// TIA Portal V17 export
// export: Created 2023-02-13T11:16:45.7840585Z, ExportSetting WithDefaults, DisplayName Totally Integrated Automation Portal, DisplayVersion V17, DisplayName TIA Portal Openness, DisplayVersion V17, DisplayName TIA Portal Teamcenter Gateway, DisplayVersion V17, DisplayName TIA Portal Version Control Interface, DisplayVersion V17, DisplayName SINAMICS Startdrive Advanced, DisplayVersion V17, DisplayName SINAMICS Startdrive G130, G150, S120, S150, SINAMICS MV, S210, DisplayVersion V17, DisplayName SINAMICS Startdrive G110M, G120, G120C, G120D, G120P, G115D, DisplayVersion V17, DisplayName STEP 7 Professional, DisplayVersion V17, DisplayName STEP 7 Safety, DisplayVersion V17, DisplayName WinCC Professional, DisplayVersion V17
ORGANIZATION_BLOCK "Totalizer_OB"   // OB31, LAD, CyclicInterrupt
{ S7_Optimized_Access := 'TRUE' }
VERSION : 0.1
// stored: AutoNumber false, IsIECCheckEnabled false, SetENOAutomatically false
   VAR_INPUT
      Initial_Call : Bool;   // Initial call of this OB
      Event_Count : Int;   // Events discarded
   END_VAR
   VAR_TEMP   // added for the SCL form of the ladder/FBD networks
      _w1 : Bool;
   END_VAR
BEGIN

REGION Network 1: Totalizer FT-00.01 Process Water Control
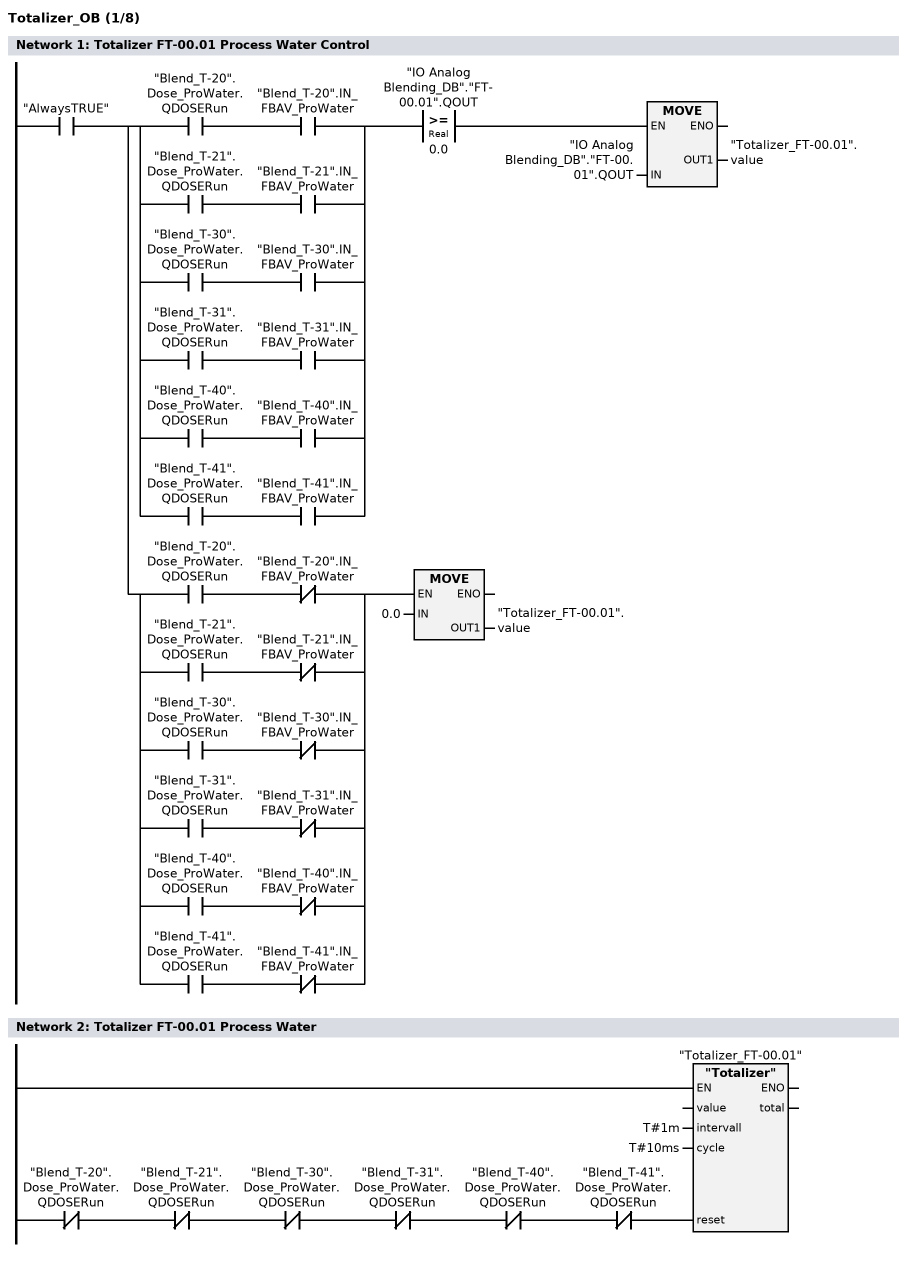
   RUNG wire#powerrail
      Contact( "AlwaysTRUE" )
      wire#w1
      Contact( "Blend_T-20".Dose_ProWater.QDOSERun )
      Contact( "Blend_T-20".IN_FBAV_ProWater )
      wire#w2
      { S7_Templates := "SrcType := Real" } GE_Contact(in1 := "IO Analog Blending_DB"."FT-00.01".QOUT, in2 := 0.0)
      Move(in := "IO Analog Blending_DB"."FT-00.01".QOUT, out1 => "Totalizer_FT-00.01".value)
   END_RUNG
   RUNG wire#w1
      Contact( "Blend_T-21".Dose_ProWater.QDOSERun )
      Contact( "Blend_T-21".IN_FBAV_ProWater )
   END_RUNG wire#w2
   RUNG wire#w1
      Contact( "Blend_T-30".Dose_ProWater.QDOSERun )
      Contact( "Blend_T-30".IN_FBAV_ProWater )
   END_RUNG wire#w2
   RUNG wire#w1
      Contact( "Blend_T-31".Dose_ProWater.QDOSERun )
      Contact( "Blend_T-31".IN_FBAV_ProWater )
   END_RUNG wire#w2
   RUNG wire#w1
      Contact( "Blend_T-40".Dose_ProWater.QDOSERun )
      Contact( "Blend_T-40".IN_FBAV_ProWater )
   END_RUNG wire#w2
   RUNG wire#w1
      Contact( "Blend_T-41".Dose_ProWater.QDOSERun )
      Contact( "Blend_T-41".IN_FBAV_ProWater )
   END_RUNG wire#w2
   RUNG wire#w1
      Contact( "Blend_T-20".Dose_ProWater.QDOSERun )
      I_Contact( "Blend_T-20".IN_FBAV_ProWater )
      wire#w3
      Move(in := 0.0, out1 => "Totalizer_FT-00.01".value)
   END_RUNG
   RUNG wire#w1
      Contact( "Blend_T-21".Dose_ProWater.QDOSERun )
      I_Contact( "Blend_T-21".IN_FBAV_ProWater )
   END_RUNG wire#w3
   RUNG wire#w1
      Contact( "Blend_T-30".Dose_ProWater.QDOSERun )
      I_Contact( "Blend_T-30".IN_FBAV_ProWater )
   END_RUNG wire#w3
   RUNG wire#w1
      Contact( "Blend_T-31".Dose_ProWater.QDOSERun )
      I_Contact( "Blend_T-31".IN_FBAV_ProWater )
   END_RUNG wire#w3
   RUNG wire#w1
      Contact( "Blend_T-40".Dose_ProWater.QDOSERun )
      I_Contact( "Blend_T-40".IN_FBAV_ProWater )
   END_RUNG wire#w3
   RUNG wire#w1
      Contact( "Blend_T-41".Dose_ProWater.QDOSERun )
      I_Contact( "Blend_T-41".IN_FBAV_ProWater )
   END_RUNG wire#w3
   // the same network as SCL:
   IF "AlwaysTRUE" AND (("Blend_T-20".Dose_ProWater.QDOSERun AND "Blend_T-20".IN_FBAV_ProWater) OR ("Blend_T-21".Dose_ProWater.QDOSERun AND "Blend_T-21".IN_FBAV_ProWater) OR ("Blend_T-30".Dose_ProWater.QDOSERun AND "Blend_T-30".IN_FBAV_ProWater) OR ("Blend_T-31".Dose_ProWater.QDOSERun AND "Blend_T-31".IN_FBAV_ProWater) OR ("Blend_T-40".Dose_ProWater.QDOSERun AND "Blend_T-40".IN_FBAV_ProWater) OR ("Blend_T-41".Dose_ProWater.QDOSERun AND "Blend_T-41".IN_FBAV_ProWater)) AND ("IO Analog Blending_DB"."FT-00.01".QOUT >= 0.0) THEN
       "Totalizer_FT-00.01".value := "IO Analog Blending_DB"."FT-00.01".QOUT;
   END_IF;
   IF "AlwaysTRUE" AND (("Blend_T-20".Dose_ProWater.QDOSERun AND NOT "Blend_T-20".IN_FBAV_ProWater) OR ("Blend_T-21".Dose_ProWater.QDOSERun AND NOT "Blend_T-21".IN_FBAV_ProWater) OR ("Blend_T-30".Dose_ProWater.QDOSERun AND NOT "Blend_T-30".IN_FBAV_ProWater) OR ("Blend_T-31".Dose_ProWater.QDOSERun AND NOT "Blend_T-31".IN_FBAV_ProWater) OR ("Blend_T-40".Dose_ProWater.QDOSERun AND NOT "Blend_T-40".IN_FBAV_ProWater) OR ("Blend_T-41".Dose_ProWater.QDOSERun AND NOT "Blend_T-41".IN_FBAV_ProWater)) THEN
       "Totalizer_FT-00.01".value := 0.0;
   END_IF;
END_REGION

REGION Network 2: Totalizer FT-00.01 Process Water
   RUNG wire#powerrail
      "Totalizer_FT-00.01"(reset := wire#w1, value :=, intervall := T#1m, cycle := T#10ms, total =>)
   END_RUNG
   RUNG wire#powerrail
      I_Contact( "Blend_T-20".Dose_ProWater.QDOSERun )
      I_Contact( "Blend_T-21".Dose_ProWater.QDOSERun )
      I_Contact( "Blend_T-30".Dose_ProWater.QDOSERun )
      I_Contact( "Blend_T-31".Dose_ProWater.QDOSERun )
      I_Contact( "Blend_T-40".Dose_ProWater.QDOSERun )
      I_Contact( "Blend_T-41".Dose_ProWater.QDOSERun )
   END_RUNG wire#w1
   // the same network as SCL:
   "Totalizer_FT-00.01"(intervall := T#1m,   // "Totalizer"
                        cycle := T#10ms,
                        reset := NOT "Blend_T-20".Dose_ProWater.QDOSERun AND NOT "Blend_T-21".Dose_ProWater.QDOSERun AND NOT "Blend_T-30".Dose_ProWater.QDOSERun AND NOT "Blend_T-31".Dose_ProWater.QDOSERun AND NOT "Blend_T-40".Dose_ProWater.QDOSERun AND NOT "Blend_T-41".Dose_ProWater.QDOSERun);
END_REGION

REGION Network 4: Totalizer FT.02.01 Chili Awetan 1 Control
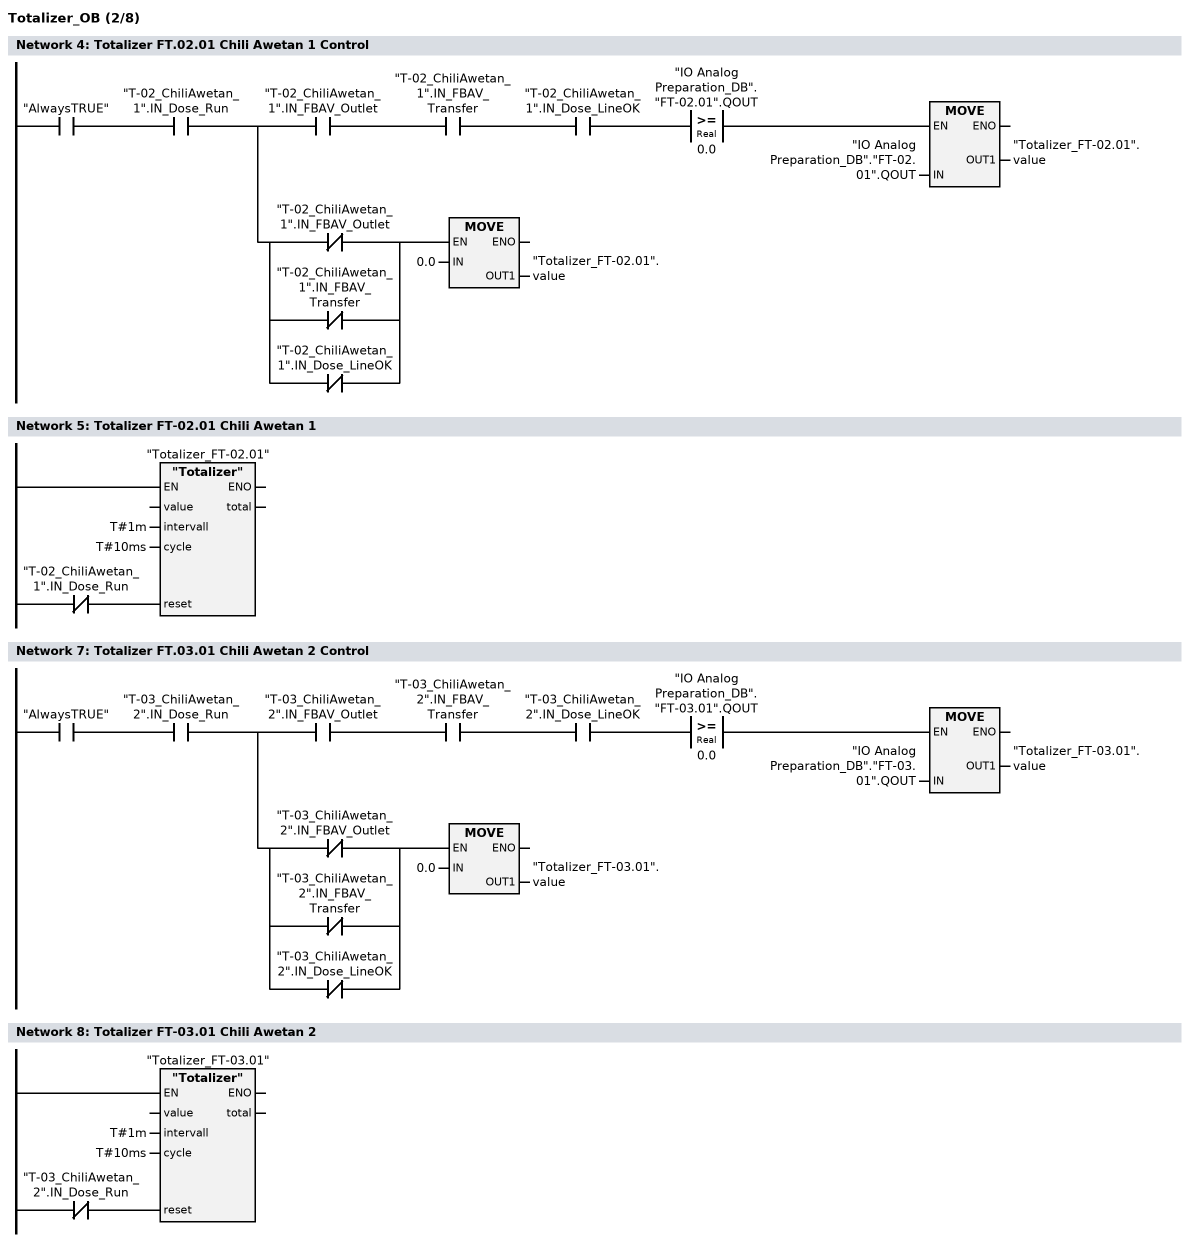
   RUNG wire#powerrail
      Contact( "AlwaysTRUE" )
      Contact( "T-02_ChiliAwetan_1".IN_Dose_Run )
      wire#w1
      Contact( "T-02_ChiliAwetan_1".IN_FBAV_Outlet )
      Contact( "T-02_ChiliAwetan_1".IN_FBAV_Transfer )
      Contact( "T-02_ChiliAwetan_1".IN_Dose_LineOK )
      { S7_Templates := "SrcType := Real" } GE_Contact(in1 := "IO Analog Preparation_DB"."FT-02.01".QOUT, in2 := 0.0)
      Move(in := "IO Analog Preparation_DB"."FT-02.01".QOUT, out1 => "Totalizer_FT-02.01".value)
   END_RUNG
   RUNG wire#w1
      I_Contact( "T-02_ChiliAwetan_1".IN_FBAV_Outlet )
      wire#w2
      Move(in := 0.0, out1 => "Totalizer_FT-02.01".value)
   END_RUNG
   RUNG wire#w1
      I_Contact( "T-02_ChiliAwetan_1".IN_FBAV_Transfer )
   END_RUNG wire#w2
   RUNG wire#w1
      I_Contact( "T-02_ChiliAwetan_1".IN_Dose_LineOK )
   END_RUNG wire#w2
   // the same network as SCL:
   #_w1 := "AlwaysTRUE" AND "T-02_ChiliAwetan_1".IN_Dose_Run;
   IF #_w1 AND "T-02_ChiliAwetan_1".IN_FBAV_Outlet AND "T-02_ChiliAwetan_1".IN_FBAV_Transfer AND "T-02_ChiliAwetan_1".IN_Dose_LineOK AND ("IO Analog Preparation_DB"."FT-02.01".QOUT >= 0.0) THEN
       "Totalizer_FT-02.01".value := "IO Analog Preparation_DB"."FT-02.01".QOUT;
   END_IF;
   IF #_w1 AND (NOT "T-02_ChiliAwetan_1".IN_FBAV_Outlet OR NOT "T-02_ChiliAwetan_1".IN_FBAV_Transfer OR NOT "T-02_ChiliAwetan_1".IN_Dose_LineOK) THEN
       "Totalizer_FT-02.01".value := 0.0;
   END_IF;
END_REGION

REGION Network 5: Totalizer FT-02.01 Chili Awetan 1
   RUNG wire#powerrail
      "Totalizer_FT-02.01"(reset := wire#w1, value :=, intervall := T#1m, cycle := T#10ms, total =>)
   END_RUNG
   RUNG wire#powerrail
      I_Contact( "T-02_ChiliAwetan_1".IN_Dose_Run )
   END_RUNG wire#w1
   // the same network as SCL:
   "Totalizer_FT-02.01"(intervall := T#1m, cycle := T#10ms, reset := NOT "T-02_ChiliAwetan_1".IN_Dose_Run);   // "Totalizer"
END_REGION

REGION Network 7: Totalizer FT.03.01 Chili Awetan 2 Control
   RUNG wire#powerrail
      Contact( "AlwaysTRUE" )
      Contact( "T-03_ChiliAwetan_2".IN_Dose_Run )
      wire#w1
      Contact( "T-03_ChiliAwetan_2".IN_FBAV_Outlet )
      Contact( "T-03_ChiliAwetan_2".IN_FBAV_Transfer )
      Contact( "T-03_ChiliAwetan_2".IN_Dose_LineOK )
      { S7_Templates := "SrcType := Real" } GE_Contact(in1 := "IO Analog Preparation_DB"."FT-03.01".QOUT, in2 := 0.0)
      Move(in := "IO Analog Preparation_DB"."FT-03.01".QOUT, out1 => "Totalizer_FT-03.01".value)
   END_RUNG
   RUNG wire#w1
      I_Contact( "T-03_ChiliAwetan_2".IN_FBAV_Outlet )
      wire#w2
      Move(in := 0.0, out1 => "Totalizer_FT-03.01".value)
   END_RUNG
   RUNG wire#w1
      I_Contact( "T-03_ChiliAwetan_2".IN_FBAV_Transfer )
   END_RUNG wire#w2
   RUNG wire#w1
      I_Contact( "T-03_ChiliAwetan_2".IN_Dose_LineOK )
   END_RUNG wire#w2
   // the same network as SCL:
   #_w1 := "AlwaysTRUE" AND "T-03_ChiliAwetan_2".IN_Dose_Run;
   IF #_w1 AND "T-03_ChiliAwetan_2".IN_FBAV_Outlet AND "T-03_ChiliAwetan_2".IN_FBAV_Transfer AND "T-03_ChiliAwetan_2".IN_Dose_LineOK AND ("IO Analog Preparation_DB"."FT-03.01".QOUT >= 0.0) THEN
       "Totalizer_FT-03.01".value := "IO Analog Preparation_DB"."FT-03.01".QOUT;
   END_IF;
   IF #_w1 AND (NOT "T-03_ChiliAwetan_2".IN_FBAV_Outlet OR NOT "T-03_ChiliAwetan_2".IN_FBAV_Transfer OR NOT "T-03_ChiliAwetan_2".IN_Dose_LineOK) THEN
       "Totalizer_FT-03.01".value := 0.0;
   END_IF;
END_REGION

REGION Network 8: Totalizer FT-03.01 Chili Awetan 2
   RUNG wire#powerrail
      "Totalizer_FT-03.01"(reset := wire#w1, value :=, intervall := T#1m, cycle := T#10ms, total =>)
   END_RUNG
   RUNG wire#powerrail
      I_Contact( "T-03_ChiliAwetan_2".IN_Dose_Run )
   END_RUNG wire#w1
   // the same network as SCL:
   "Totalizer_FT-03.01"(intervall := T#1m, cycle := T#10ms, reset := NOT "T-03_ChiliAwetan_2".IN_Dose_Run);   // "Totalizer"
END_REGION

REGION Network 10: Totalizer FT.04.01 Chili Awetan 3 Control
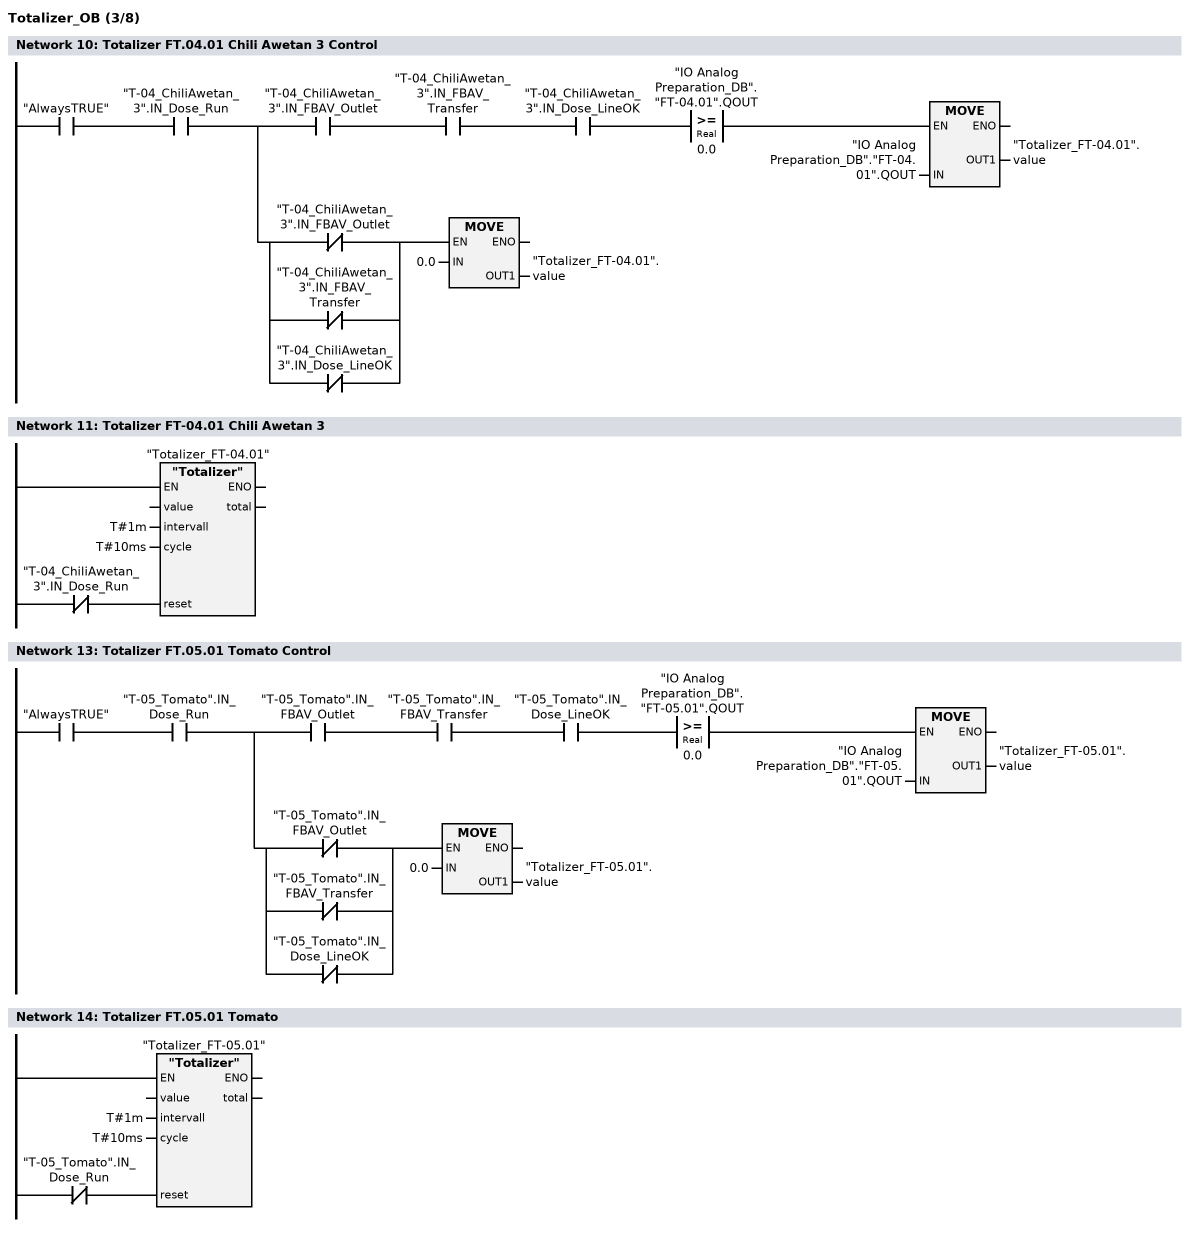
   RUNG wire#powerrail
      Contact( "AlwaysTRUE" )
      Contact( "T-04_ChiliAwetan_3".IN_Dose_Run )
      wire#w1
      Contact( "T-04_ChiliAwetan_3".IN_FBAV_Outlet )
      Contact( "T-04_ChiliAwetan_3".IN_FBAV_Transfer )
      Contact( "T-04_ChiliAwetan_3".IN_Dose_LineOK )
      { S7_Templates := "SrcType := Real" } GE_Contact(in1 := "IO Analog Preparation_DB"."FT-04.01".QOUT, in2 := 0.0)
      Move(in := "IO Analog Preparation_DB"."FT-04.01".QOUT, out1 => "Totalizer_FT-04.01".value)
   END_RUNG
   RUNG wire#w1
      I_Contact( "T-04_ChiliAwetan_3".IN_FBAV_Outlet )
      wire#w2
      Move(in := 0.0, out1 => "Totalizer_FT-04.01".value)
   END_RUNG
   RUNG wire#w1
      I_Contact( "T-04_ChiliAwetan_3".IN_FBAV_Transfer )
   END_RUNG wire#w2
   RUNG wire#w1
      I_Contact( "T-04_ChiliAwetan_3".IN_Dose_LineOK )
   END_RUNG wire#w2
   // the same network as SCL:
   #_w1 := "AlwaysTRUE" AND "T-04_ChiliAwetan_3".IN_Dose_Run;
   IF #_w1 AND "T-04_ChiliAwetan_3".IN_FBAV_Outlet AND "T-04_ChiliAwetan_3".IN_FBAV_Transfer AND "T-04_ChiliAwetan_3".IN_Dose_LineOK AND ("IO Analog Preparation_DB"."FT-04.01".QOUT >= 0.0) THEN
       "Totalizer_FT-04.01".value := "IO Analog Preparation_DB"."FT-04.01".QOUT;
   END_IF;
   IF #_w1 AND (NOT "T-04_ChiliAwetan_3".IN_FBAV_Outlet OR NOT "T-04_ChiliAwetan_3".IN_FBAV_Transfer OR NOT "T-04_ChiliAwetan_3".IN_Dose_LineOK) THEN
       "Totalizer_FT-04.01".value := 0.0;
   END_IF;
END_REGION

REGION Network 11: Totalizer FT-04.01 Chili Awetan 3
   RUNG wire#powerrail
      "Totalizer_FT-04.01"(reset := wire#w1, value :=, intervall := T#1m, cycle := T#10ms, total =>)
   END_RUNG
   RUNG wire#powerrail
      I_Contact( "T-04_ChiliAwetan_3".IN_Dose_Run )
   END_RUNG wire#w1
   // the same network as SCL:
   "Totalizer_FT-04.01"(intervall := T#1m, cycle := T#10ms, reset := NOT "T-04_ChiliAwetan_3".IN_Dose_Run);   // "Totalizer"
END_REGION

REGION Network 13: Totalizer FT.05.01 Tomato Control
   RUNG wire#powerrail
      Contact( "AlwaysTRUE" )
      Contact( "T-05_Tomato".IN_Dose_Run )
      wire#w1
      Contact( "T-05_Tomato".IN_FBAV_Outlet )
      Contact( "T-05_Tomato".IN_FBAV_Transfer )
      Contact( "T-05_Tomato".IN_Dose_LineOK )
      { S7_Templates := "SrcType := Real" } GE_Contact(in1 := "IO Analog Preparation_DB"."FT-05.01".QOUT, in2 := 0.0)
      Move(in := "IO Analog Preparation_DB"."FT-05.01".QOUT, out1 => "Totalizer_FT-05.01".value)
   END_RUNG
   RUNG wire#w1
      I_Contact( "T-05_Tomato".IN_FBAV_Outlet )
      wire#w2
      Move(in := 0.0, out1 => "Totalizer_FT-05.01".value)
   END_RUNG
   RUNG wire#w1
      I_Contact( "T-05_Tomato".IN_FBAV_Transfer )
   END_RUNG wire#w2
   RUNG wire#w1
      I_Contact( "T-05_Tomato".IN_Dose_LineOK )
   END_RUNG wire#w2
   // the same network as SCL:
   #_w1 := "AlwaysTRUE" AND "T-05_Tomato".IN_Dose_Run;
   IF #_w1 AND "T-05_Tomato".IN_FBAV_Outlet AND "T-05_Tomato".IN_FBAV_Transfer AND "T-05_Tomato".IN_Dose_LineOK AND ("IO Analog Preparation_DB"."FT-05.01".QOUT >= 0.0) THEN
       "Totalizer_FT-05.01".value := "IO Analog Preparation_DB"."FT-05.01".QOUT;
   END_IF;
   IF #_w1 AND (NOT "T-05_Tomato".IN_FBAV_Outlet OR NOT "T-05_Tomato".IN_FBAV_Transfer OR NOT "T-05_Tomato".IN_Dose_LineOK) THEN
       "Totalizer_FT-05.01".value := 0.0;
   END_IF;
END_REGION

REGION Network 14: Totalizer FT.05.01 Tomato
   RUNG wire#powerrail
      "Totalizer_FT-05.01"(reset := wire#w1, value :=, intervall := T#1m, cycle := T#10ms, total =>)
   END_RUNG
   RUNG wire#powerrail
      I_Contact( "T-05_Tomato".IN_Dose_Run )
   END_RUNG wire#w1
   // the same network as SCL:
   "Totalizer_FT-05.01"(intervall := T#1m, cycle := T#10ms, reset := NOT "T-05_Tomato".IN_Dose_Run);   // "Totalizer"
END_REGION

REGION Network 16: Totalizer FT.06.01 Chili Fresh 1 Control
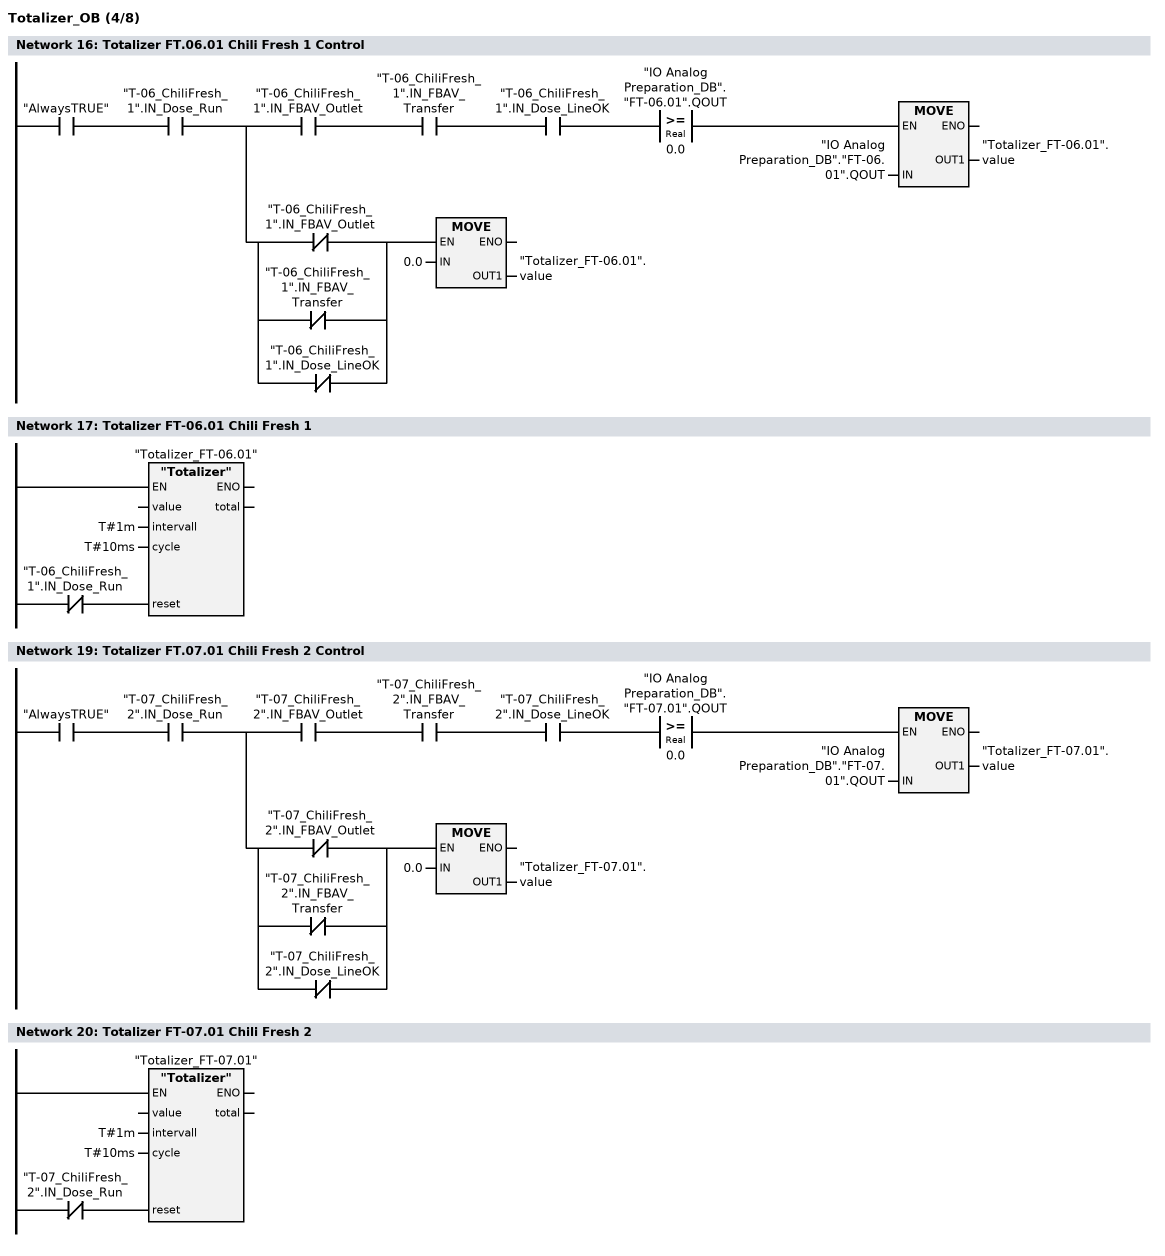
   RUNG wire#powerrail
      Contact( "AlwaysTRUE" )
      Contact( "T-06_ChiliFresh_1".IN_Dose_Run )
      wire#w1
      Contact( "T-06_ChiliFresh_1".IN_FBAV_Outlet )
      Contact( "T-06_ChiliFresh_1".IN_FBAV_Transfer )
      Contact( "T-06_ChiliFresh_1".IN_Dose_LineOK )
      { S7_Templates := "SrcType := Real" } GE_Contact(in1 := "IO Analog Preparation_DB"."FT-06.01".QOUT, in2 := 0.0)
      Move(in := "IO Analog Preparation_DB"."FT-06.01".QOUT, out1 => "Totalizer_FT-06.01".value)
   END_RUNG
   RUNG wire#w1
      I_Contact( "T-06_ChiliFresh_1".IN_FBAV_Outlet )
      wire#w2
      Move(in := 0.0, out1 => "Totalizer_FT-06.01".value)
   END_RUNG
   RUNG wire#w1
      I_Contact( "T-06_ChiliFresh_1".IN_FBAV_Transfer )
   END_RUNG wire#w2
   RUNG wire#w1
      I_Contact( "T-06_ChiliFresh_1".IN_Dose_LineOK )
   END_RUNG wire#w2
   // the same network as SCL:
   #_w1 := "AlwaysTRUE" AND "T-06_ChiliFresh_1".IN_Dose_Run;
   IF #_w1 AND "T-06_ChiliFresh_1".IN_FBAV_Outlet AND "T-06_ChiliFresh_1".IN_FBAV_Transfer AND "T-06_ChiliFresh_1".IN_Dose_LineOK AND ("IO Analog Preparation_DB"."FT-06.01".QOUT >= 0.0) THEN
       "Totalizer_FT-06.01".value := "IO Analog Preparation_DB"."FT-06.01".QOUT;
   END_IF;
   IF #_w1 AND (NOT "T-06_ChiliFresh_1".IN_FBAV_Outlet OR NOT "T-06_ChiliFresh_1".IN_FBAV_Transfer OR NOT "T-06_ChiliFresh_1".IN_Dose_LineOK) THEN
       "Totalizer_FT-06.01".value := 0.0;
   END_IF;
END_REGION

REGION Network 17: Totalizer FT-06.01 Chili Fresh 1
   RUNG wire#powerrail
      "Totalizer_FT-06.01"(reset := wire#w1, value :=, intervall := T#1m, cycle := T#10ms, total =>)
   END_RUNG
   RUNG wire#powerrail
      I_Contact( "T-06_ChiliFresh_1".IN_Dose_Run )
   END_RUNG wire#w1
   // the same network as SCL:
   "Totalizer_FT-06.01"(intervall := T#1m, cycle := T#10ms, reset := NOT "T-06_ChiliFresh_1".IN_Dose_Run);   // "Totalizer"
END_REGION

REGION Network 19: Totalizer FT.07.01 Chili Fresh 2 Control
   RUNG wire#powerrail
      Contact( "AlwaysTRUE" )
      Contact( "T-07_ChiliFresh_2".IN_Dose_Run )
      wire#w1
      Contact( "T-07_ChiliFresh_2".IN_FBAV_Outlet )
      Contact( "T-07_ChiliFresh_2".IN_FBAV_Transfer )
      Contact( "T-07_ChiliFresh_2".IN_Dose_LineOK )
      { S7_Templates := "SrcType := Real" } GE_Contact(in1 := "IO Analog Preparation_DB"."FT-07.01".QOUT, in2 := 0.0)
      Move(in := "IO Analog Preparation_DB"."FT-07.01".QOUT, out1 => "Totalizer_FT-07.01".value)
   END_RUNG
   RUNG wire#w1
      I_Contact( "T-07_ChiliFresh_2".IN_FBAV_Outlet )
      wire#w2
      Move(in := 0.0, out1 => "Totalizer_FT-07.01".value)
   END_RUNG
   RUNG wire#w1
      I_Contact( "T-07_ChiliFresh_2".IN_FBAV_Transfer )
   END_RUNG wire#w2
   RUNG wire#w1
      I_Contact( "T-07_ChiliFresh_2".IN_Dose_LineOK )
   END_RUNG wire#w2
   // the same network as SCL:
   #_w1 := "AlwaysTRUE" AND "T-07_ChiliFresh_2".IN_Dose_Run;
   IF #_w1 AND "T-07_ChiliFresh_2".IN_FBAV_Outlet AND "T-07_ChiliFresh_2".IN_FBAV_Transfer AND "T-07_ChiliFresh_2".IN_Dose_LineOK AND ("IO Analog Preparation_DB"."FT-07.01".QOUT >= 0.0) THEN
       "Totalizer_FT-07.01".value := "IO Analog Preparation_DB"."FT-07.01".QOUT;
   END_IF;
   IF #_w1 AND (NOT "T-07_ChiliFresh_2".IN_FBAV_Outlet OR NOT "T-07_ChiliFresh_2".IN_FBAV_Transfer OR NOT "T-07_ChiliFresh_2".IN_Dose_LineOK) THEN
       "Totalizer_FT-07.01".value := 0.0;
   END_IF;
END_REGION

REGION Network 20: Totalizer FT-07.01 Chili Fresh 2
   RUNG wire#powerrail
      "Totalizer_FT-07.01"(reset := wire#w1, value :=, intervall := T#1m, cycle := T#10ms, total =>)
   END_RUNG
   RUNG wire#powerrail
      I_Contact( "T-07_ChiliFresh_2".IN_Dose_Run )
   END_RUNG wire#w1
   // the same network as SCL:
   "Totalizer_FT-07.01"(intervall := T#1m, cycle := T#10ms, reset := NOT "T-07_ChiliFresh_2".IN_Dose_Run);   // "Totalizer"
END_REGION

REGION Network 22: Totalizer FT.08.01 Chili Fresh 3 Control
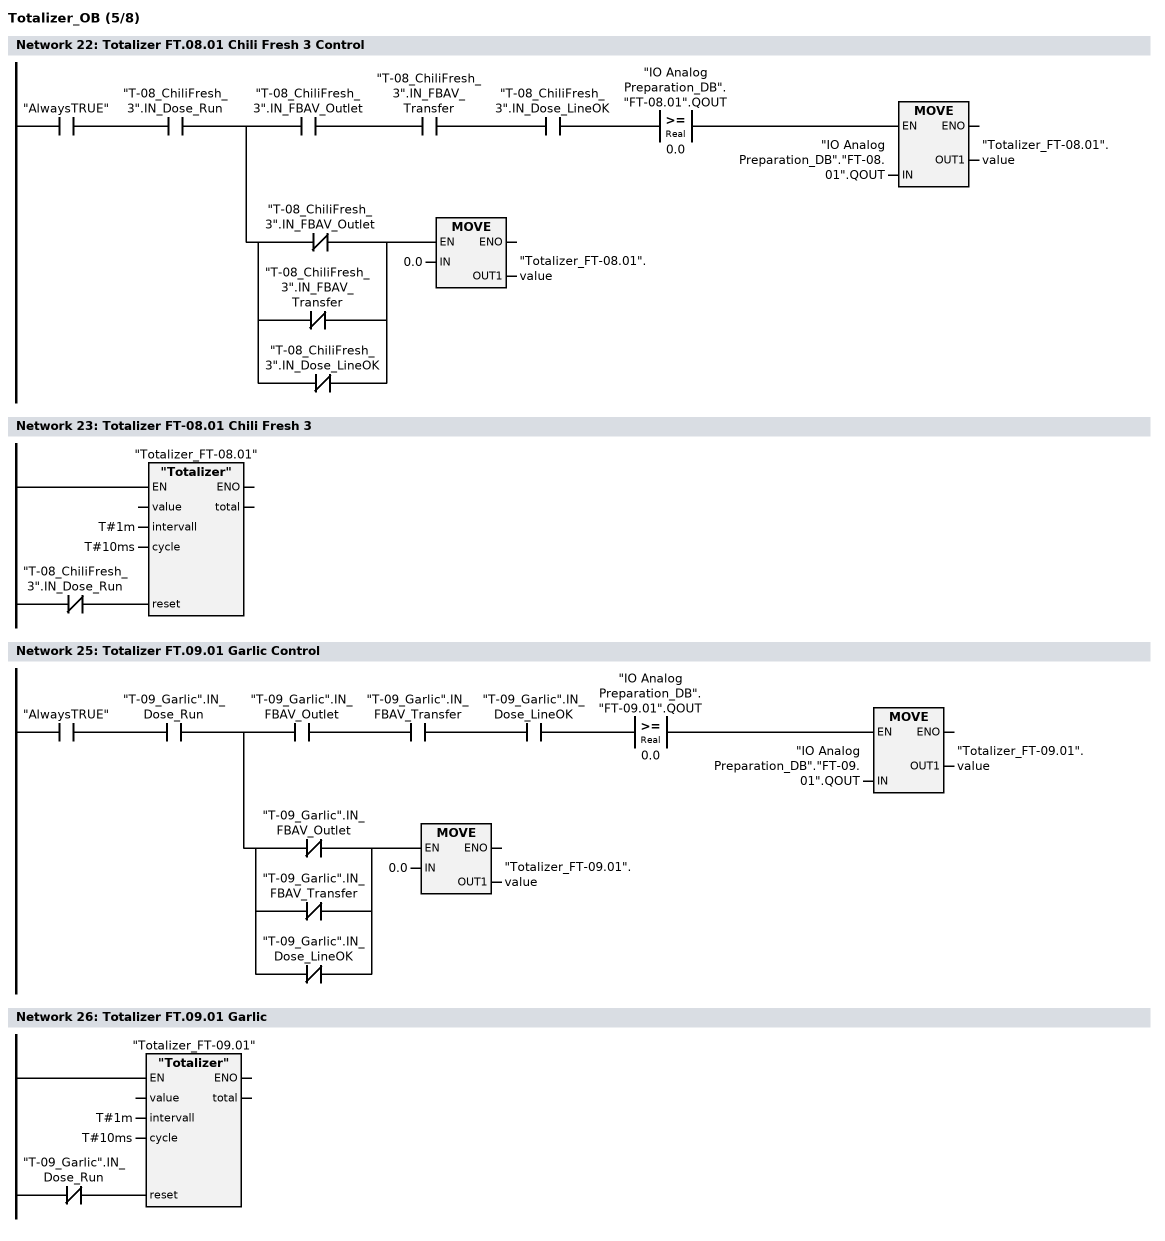
   RUNG wire#powerrail
      Contact( "AlwaysTRUE" )
      Contact( "T-08_ChiliFresh_3".IN_Dose_Run )
      wire#w1
      Contact( "T-08_ChiliFresh_3".IN_FBAV_Outlet )
      Contact( "T-08_ChiliFresh_3".IN_FBAV_Transfer )
      Contact( "T-08_ChiliFresh_3".IN_Dose_LineOK )
      { S7_Templates := "SrcType := Real" } GE_Contact(in1 := "IO Analog Preparation_DB"."FT-08.01".QOUT, in2 := 0.0)
      Move(in := "IO Analog Preparation_DB"."FT-08.01".QOUT, out1 => "Totalizer_FT-08.01".value)
   END_RUNG
   RUNG wire#w1
      I_Contact( "T-08_ChiliFresh_3".IN_FBAV_Outlet )
      wire#w2
      Move(in := 0.0, out1 => "Totalizer_FT-08.01".value)
   END_RUNG
   RUNG wire#w1
      I_Contact( "T-08_ChiliFresh_3".IN_FBAV_Transfer )
   END_RUNG wire#w2
   RUNG wire#w1
      I_Contact( "T-08_ChiliFresh_3".IN_Dose_LineOK )
   END_RUNG wire#w2
   // the same network as SCL:
   #_w1 := "AlwaysTRUE" AND "T-08_ChiliFresh_3".IN_Dose_Run;
   IF #_w1 AND "T-08_ChiliFresh_3".IN_FBAV_Outlet AND "T-08_ChiliFresh_3".IN_FBAV_Transfer AND "T-08_ChiliFresh_3".IN_Dose_LineOK AND ("IO Analog Preparation_DB"."FT-08.01".QOUT >= 0.0) THEN
       "Totalizer_FT-08.01".value := "IO Analog Preparation_DB"."FT-08.01".QOUT;
   END_IF;
   IF #_w1 AND (NOT "T-08_ChiliFresh_3".IN_FBAV_Outlet OR NOT "T-08_ChiliFresh_3".IN_FBAV_Transfer OR NOT "T-08_ChiliFresh_3".IN_Dose_LineOK) THEN
       "Totalizer_FT-08.01".value := 0.0;
   END_IF;
END_REGION

REGION Network 23: Totalizer FT-08.01 Chili Fresh 3
   RUNG wire#powerrail
      "Totalizer_FT-08.01"(reset := wire#w1, value :=, intervall := T#1m, cycle := T#10ms, total =>)
   END_RUNG
   RUNG wire#powerrail
      I_Contact( "T-08_ChiliFresh_3".IN_Dose_Run )
   END_RUNG wire#w1
   // the same network as SCL:
   "Totalizer_FT-08.01"(intervall := T#1m, cycle := T#10ms, reset := NOT "T-08_ChiliFresh_3".IN_Dose_Run);   // "Totalizer"
END_REGION

REGION Network 25: Totalizer FT.09.01 Garlic Control
   RUNG wire#powerrail
      Contact( "AlwaysTRUE" )
      Contact( "T-09_Garlic".IN_Dose_Run )
      wire#w1
      Contact( "T-09_Garlic".IN_FBAV_Outlet )
      Contact( "T-09_Garlic".IN_FBAV_Transfer )
      Contact( "T-09_Garlic".IN_Dose_LineOK )
      { S7_Templates := "SrcType := Real" } GE_Contact(in1 := "IO Analog Preparation_DB"."FT-09.01".QOUT, in2 := 0.0)
      Move(in := "IO Analog Preparation_DB"."FT-09.01".QOUT, out1 => "Totalizer_FT-09.01".value)
   END_RUNG
   RUNG wire#w1
      I_Contact( "T-09_Garlic".IN_FBAV_Outlet )
      wire#w2
      Move(in := 0.0, out1 => "Totalizer_FT-09.01".value)
   END_RUNG
   RUNG wire#w1
      I_Contact( "T-09_Garlic".IN_FBAV_Transfer )
   END_RUNG wire#w2
   RUNG wire#w1
      I_Contact( "T-09_Garlic".IN_Dose_LineOK )
   END_RUNG wire#w2
   // the same network as SCL:
   #_w1 := "AlwaysTRUE" AND "T-09_Garlic".IN_Dose_Run;
   IF #_w1 AND "T-09_Garlic".IN_FBAV_Outlet AND "T-09_Garlic".IN_FBAV_Transfer AND "T-09_Garlic".IN_Dose_LineOK AND ("IO Analog Preparation_DB"."FT-09.01".QOUT >= 0.0) THEN
       "Totalizer_FT-09.01".value := "IO Analog Preparation_DB"."FT-09.01".QOUT;
   END_IF;
   IF #_w1 AND (NOT "T-09_Garlic".IN_FBAV_Outlet OR NOT "T-09_Garlic".IN_FBAV_Transfer OR NOT "T-09_Garlic".IN_Dose_LineOK) THEN
       "Totalizer_FT-09.01".value := 0.0;
   END_IF;
END_REGION

REGION Network 26: Totalizer FT.09.01 Garlic
   RUNG wire#powerrail
      "Totalizer_FT-09.01"(reset := wire#w1, value :=, intervall := T#1m, cycle := T#10ms, total =>)
   END_RUNG
   RUNG wire#powerrail
      I_Contact( "T-09_Garlic".IN_Dose_Run )
   END_RUNG wire#w1
   // the same network as SCL:
   "Totalizer_FT-09.01"(intervall := T#1m, cycle := T#10ms, reset := NOT "T-09_Garlic".IN_Dose_Run);   // "Totalizer"
END_REGION

REGION Network 28: Totalizer FT.10.01 Vinegar Control
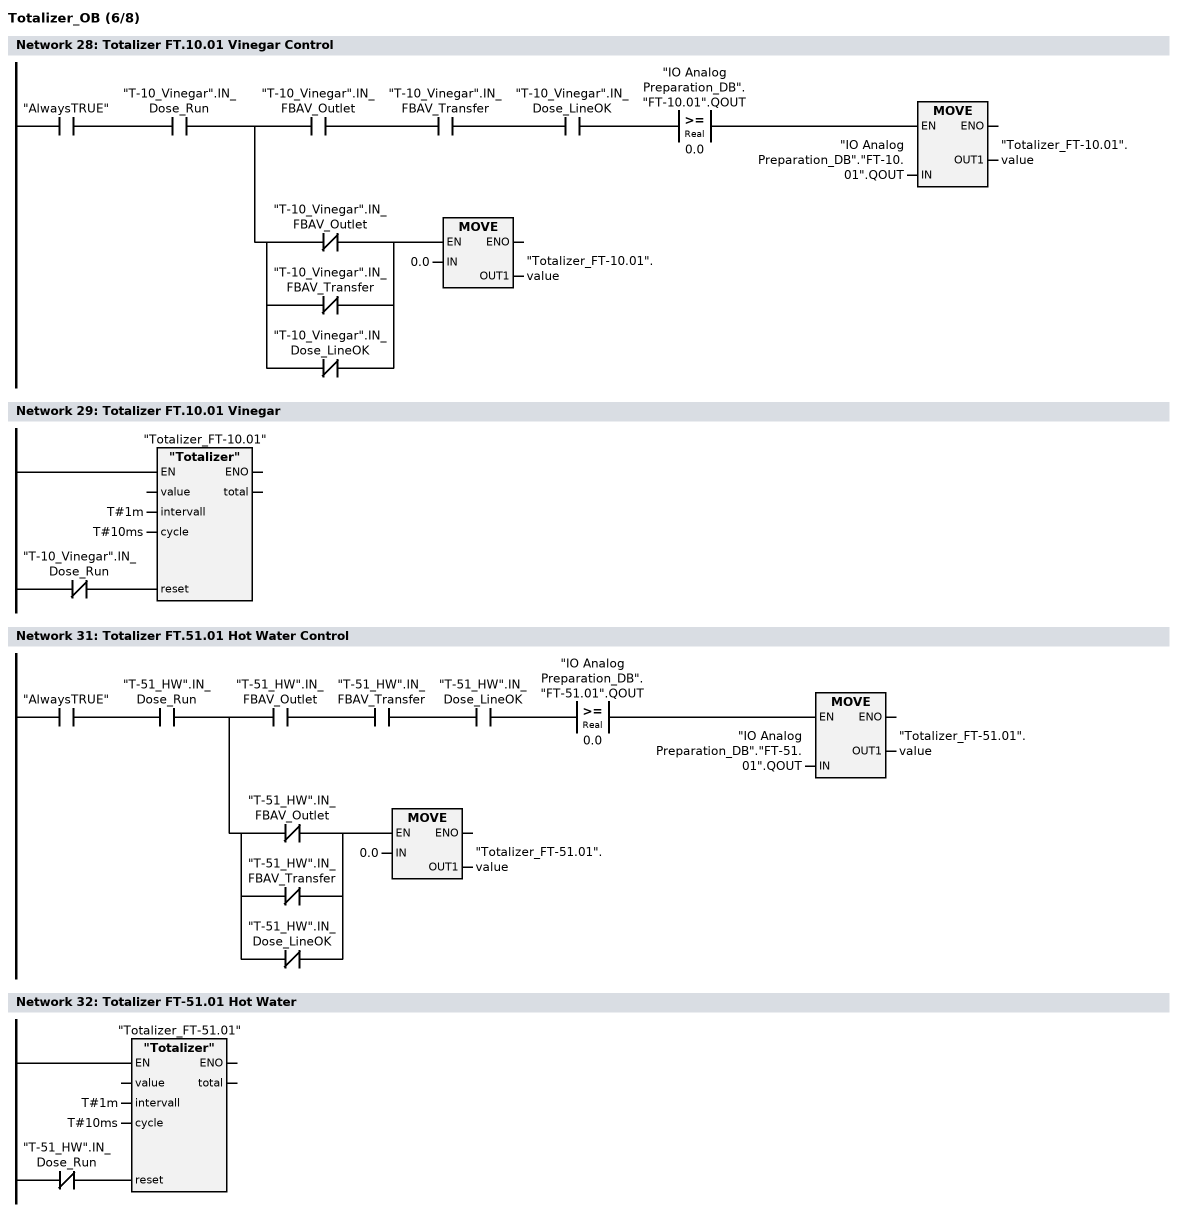
   RUNG wire#powerrail
      Contact( "AlwaysTRUE" )
      Contact( "T-10_Vinegar".IN_Dose_Run )
      wire#w1
      Contact( "T-10_Vinegar".IN_FBAV_Outlet )
      Contact( "T-10_Vinegar".IN_FBAV_Transfer )
      Contact( "T-10_Vinegar".IN_Dose_LineOK )
      { S7_Templates := "SrcType := Real" } GE_Contact(in1 := "IO Analog Preparation_DB"."FT-10.01".QOUT, in2 := 0.0)
      Move(in := "IO Analog Preparation_DB"."FT-10.01".QOUT, out1 => "Totalizer_FT-10.01".value)
   END_RUNG
   RUNG wire#w1
      I_Contact( "T-10_Vinegar".IN_FBAV_Outlet )
      wire#w2
      Move(in := 0.0, out1 => "Totalizer_FT-10.01".value)
   END_RUNG
   RUNG wire#w1
      I_Contact( "T-10_Vinegar".IN_FBAV_Transfer )
   END_RUNG wire#w2
   RUNG wire#w1
      I_Contact( "T-10_Vinegar".IN_Dose_LineOK )
   END_RUNG wire#w2
   // the same network as SCL:
   #_w1 := "AlwaysTRUE" AND "T-10_Vinegar".IN_Dose_Run;
   IF #_w1 AND "T-10_Vinegar".IN_FBAV_Outlet AND "T-10_Vinegar".IN_FBAV_Transfer AND "T-10_Vinegar".IN_Dose_LineOK AND ("IO Analog Preparation_DB"."FT-10.01".QOUT >= 0.0) THEN
       "Totalizer_FT-10.01".value := "IO Analog Preparation_DB"."FT-10.01".QOUT;
   END_IF;
   IF #_w1 AND (NOT "T-10_Vinegar".IN_FBAV_Outlet OR NOT "T-10_Vinegar".IN_FBAV_Transfer OR NOT "T-10_Vinegar".IN_Dose_LineOK) THEN
       "Totalizer_FT-10.01".value := 0.0;
   END_IF;
END_REGION

REGION Network 29: Totalizer FT.10.01 Vinegar
   RUNG wire#powerrail
      "Totalizer_FT-10.01"(reset := wire#w1, value :=, intervall := T#1m, cycle := T#10ms, total =>)
   END_RUNG
   RUNG wire#powerrail
      I_Contact( "T-10_Vinegar".IN_Dose_Run )
   END_RUNG wire#w1
   // the same network as SCL:
   "Totalizer_FT-10.01"(intervall := T#1m, cycle := T#10ms, reset := NOT "T-10_Vinegar".IN_Dose_Run);   // "Totalizer"
END_REGION

REGION Network 31: Totalizer FT.51.01 Hot Water Control
   RUNG wire#powerrail
      Contact( "AlwaysTRUE" )
      Contact( "T-51_HW".IN_Dose_Run )
      wire#w1
      Contact( "T-51_HW".IN_FBAV_Outlet )
      Contact( "T-51_HW".IN_FBAV_Transfer )
      Contact( "T-51_HW".IN_Dose_LineOK )
      { S7_Templates := "SrcType := Real" } GE_Contact(in1 := "IO Analog Preparation_DB"."FT-51.01".QOUT, in2 := 0.0)
      Move(in := "IO Analog Preparation_DB"."FT-51.01".QOUT, out1 => "Totalizer_FT-51.01".value)
   END_RUNG
   RUNG wire#w1
      I_Contact( "T-51_HW".IN_FBAV_Outlet )
      wire#w2
      Move(in := 0.0, out1 => "Totalizer_FT-51.01".value)
   END_RUNG
   RUNG wire#w1
      I_Contact( "T-51_HW".IN_FBAV_Transfer )
   END_RUNG wire#w2
   RUNG wire#w1
      I_Contact( "T-51_HW".IN_Dose_LineOK )
   END_RUNG wire#w2
   // the same network as SCL:
   #_w1 := "AlwaysTRUE" AND "T-51_HW".IN_Dose_Run;
   IF #_w1 AND "T-51_HW".IN_FBAV_Outlet AND "T-51_HW".IN_FBAV_Transfer AND "T-51_HW".IN_Dose_LineOK AND ("IO Analog Preparation_DB"."FT-51.01".QOUT >= 0.0) THEN
       "Totalizer_FT-51.01".value := "IO Analog Preparation_DB"."FT-51.01".QOUT;
   END_IF;
   IF #_w1 AND (NOT "T-51_HW".IN_FBAV_Outlet OR NOT "T-51_HW".IN_FBAV_Transfer OR NOT "T-51_HW".IN_Dose_LineOK) THEN
       "Totalizer_FT-51.01".value := 0.0;
   END_IF;
END_REGION

REGION Network 32: Totalizer FT-51.01 Hot Water
   RUNG wire#powerrail
      "Totalizer_FT-51.01"(reset := wire#w1, value :=, intervall := T#1m, cycle := T#10ms, total =>)
   END_RUNG
   RUNG wire#powerrail
      I_Contact( "T-51_HW".IN_Dose_Run )
   END_RUNG wire#w1
   // the same network as SCL:
   "Totalizer_FT-51.01"(intervall := T#1m, cycle := T#10ms, reset := NOT "T-51_HW".IN_Dose_Run);   // "Totalizer"
END_REGION

REGION Network 34: Totalizer FT-12.01 ProWater Homomixer Control
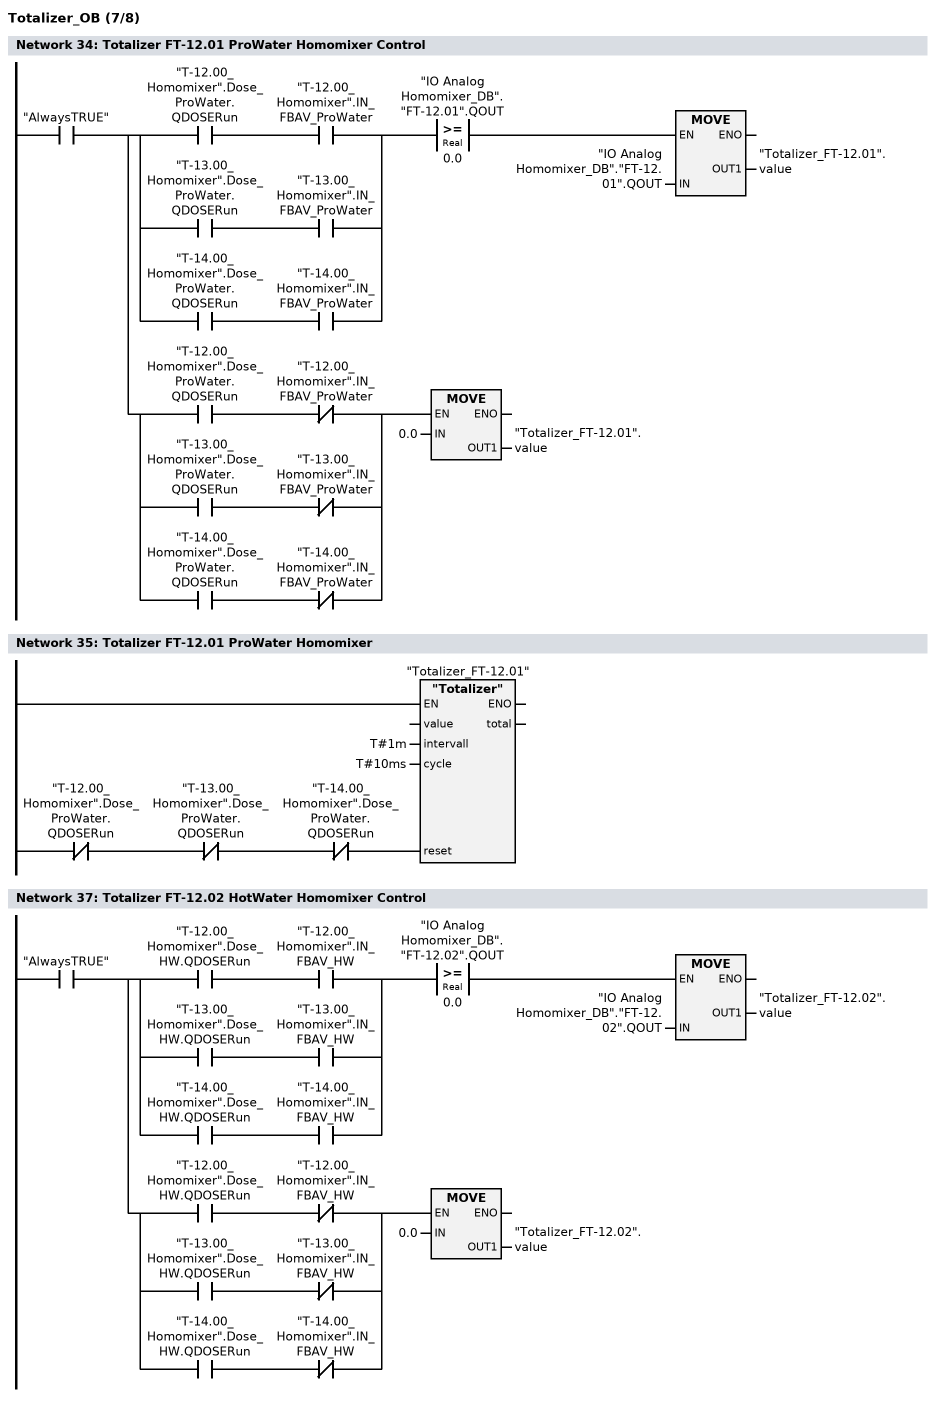
   RUNG wire#powerrail
      Contact( "AlwaysTRUE" )
      wire#w1
      Contact( "T-12.00_Homomixer".Dose_ProWater.QDOSERun )
      Contact( "T-12.00_Homomixer".IN_FBAV_ProWater )
      wire#w2
      { S7_Templates := "SrcType := Real" } GE_Contact(in1 := "IO Analog Homomixer_DB"."FT-12.01".QOUT, in2 := 0.0)
      Move(in := "IO Analog Homomixer_DB"."FT-12.01".QOUT, out1 => "Totalizer_FT-12.01".value)
   END_RUNG
   RUNG wire#w1
      Contact( "T-13.00_Homomixer".Dose_ProWater.QDOSERun )
      Contact( "T-13.00_Homomixer".IN_FBAV_ProWater )
   END_RUNG wire#w2
   RUNG wire#w1
      Contact( "T-14.00_Homomixer".Dose_ProWater.QDOSERun )
      Contact( "T-14.00_Homomixer".IN_FBAV_ProWater )
   END_RUNG wire#w2
   RUNG wire#w1
      Contact( "T-12.00_Homomixer".Dose_ProWater.QDOSERun )
      I_Contact( "T-12.00_Homomixer".IN_FBAV_ProWater )
      wire#w3
      Move(in := 0.0, out1 => "Totalizer_FT-12.01".value)
   END_RUNG
   RUNG wire#w1
      Contact( "T-13.00_Homomixer".Dose_ProWater.QDOSERun )
      I_Contact( "T-13.00_Homomixer".IN_FBAV_ProWater )
   END_RUNG wire#w3
   RUNG wire#w1
      Contact( "T-14.00_Homomixer".Dose_ProWater.QDOSERun )
      I_Contact( "T-14.00_Homomixer".IN_FBAV_ProWater )
   END_RUNG wire#w3
   // the same network as SCL:
   IF "AlwaysTRUE" AND (("T-12.00_Homomixer".Dose_ProWater.QDOSERun AND "T-12.00_Homomixer".IN_FBAV_ProWater) OR ("T-13.00_Homomixer".Dose_ProWater.QDOSERun AND "T-13.00_Homomixer".IN_FBAV_ProWater) OR ("T-14.00_Homomixer".Dose_ProWater.QDOSERun AND "T-14.00_Homomixer".IN_FBAV_ProWater)) AND ("IO Analog Homomixer_DB"."FT-12.01".QOUT >= 0.0) THEN
       "Totalizer_FT-12.01".value := "IO Analog Homomixer_DB"."FT-12.01".QOUT;
   END_IF;
   IF "AlwaysTRUE" AND (("T-12.00_Homomixer".Dose_ProWater.QDOSERun AND NOT "T-12.00_Homomixer".IN_FBAV_ProWater) OR ("T-13.00_Homomixer".Dose_ProWater.QDOSERun AND NOT "T-13.00_Homomixer".IN_FBAV_ProWater) OR ("T-14.00_Homomixer".Dose_ProWater.QDOSERun AND NOT "T-14.00_Homomixer".IN_FBAV_ProWater)) THEN
       "Totalizer_FT-12.01".value := 0.0;
   END_IF;
END_REGION

REGION Network 35: Totalizer FT-12.01 ProWater Homomixer
   RUNG wire#powerrail
      "Totalizer_FT-12.01"(reset := wire#w1, value :=, intervall := T#1m, cycle := T#10ms, total =>)
   END_RUNG
   RUNG wire#powerrail
      I_Contact( "T-12.00_Homomixer".Dose_ProWater.QDOSERun )
      I_Contact( "T-13.00_Homomixer".Dose_ProWater.QDOSERun )
      I_Contact( "T-14.00_Homomixer".Dose_ProWater.QDOSERun )
   END_RUNG wire#w1
   // the same network as SCL:
   "Totalizer_FT-12.01"(intervall := T#1m,   // "Totalizer"
                        cycle := T#10ms,
                        reset := NOT "T-12.00_Homomixer".Dose_ProWater.QDOSERun AND NOT "T-13.00_Homomixer".Dose_ProWater.QDOSERun AND NOT "T-14.00_Homomixer".Dose_ProWater.QDOSERun);
END_REGION

REGION Network 37: Totalizer FT-12.02 HotWater Homomixer Control
   RUNG wire#powerrail
      Contact( "AlwaysTRUE" )
      wire#w1
      Contact( "T-12.00_Homomixer".Dose_HW.QDOSERun )
      Contact( "T-12.00_Homomixer".IN_FBAV_HW )
      wire#w2
      { S7_Templates := "SrcType := Real" } GE_Contact(in1 := "IO Analog Homomixer_DB"."FT-12.02".QOUT, in2 := 0.0)
      Move(in := "IO Analog Homomixer_DB"."FT-12.02".QOUT, out1 => "Totalizer_FT-12.02".value)
   END_RUNG
   RUNG wire#w1
      Contact( "T-13.00_Homomixer".Dose_HW.QDOSERun )
      Contact( "T-13.00_Homomixer".IN_FBAV_HW )
   END_RUNG wire#w2
   RUNG wire#w1
      Contact( "T-14.00_Homomixer".Dose_HW.QDOSERun )
      Contact( "T-14.00_Homomixer".IN_FBAV_HW )
   END_RUNG wire#w2
   RUNG wire#w1
      Contact( "T-12.00_Homomixer".Dose_HW.QDOSERun )
      I_Contact( "T-12.00_Homomixer".IN_FBAV_HW )
      wire#w3
      Move(in := 0.0, out1 => "Totalizer_FT-12.02".value)
   END_RUNG
   RUNG wire#w1
      Contact( "T-13.00_Homomixer".Dose_HW.QDOSERun )
      I_Contact( "T-13.00_Homomixer".IN_FBAV_HW )
   END_RUNG wire#w3
   RUNG wire#w1
      Contact( "T-14.00_Homomixer".Dose_HW.QDOSERun )
      I_Contact( "T-14.00_Homomixer".IN_FBAV_HW )
   END_RUNG wire#w3
   // the same network as SCL:
   IF "AlwaysTRUE" AND (("T-12.00_Homomixer".Dose_HW.QDOSERun AND "T-12.00_Homomixer".IN_FBAV_HW) OR ("T-13.00_Homomixer".Dose_HW.QDOSERun AND "T-13.00_Homomixer".IN_FBAV_HW) OR ("T-14.00_Homomixer".Dose_HW.QDOSERun AND "T-14.00_Homomixer".IN_FBAV_HW)) AND ("IO Analog Homomixer_DB"."FT-12.02".QOUT >= 0.0) THEN
       "Totalizer_FT-12.02".value := "IO Analog Homomixer_DB"."FT-12.02".QOUT;
   END_IF;
   IF "AlwaysTRUE" AND (("T-12.00_Homomixer".Dose_HW.QDOSERun AND NOT "T-12.00_Homomixer".IN_FBAV_HW) OR ("T-13.00_Homomixer".Dose_HW.QDOSERun AND NOT "T-13.00_Homomixer".IN_FBAV_HW) OR ("T-14.00_Homomixer".Dose_HW.QDOSERun AND NOT "T-14.00_Homomixer".IN_FBAV_HW)) THEN
       "Totalizer_FT-12.02".value := 0.0;
   END_IF;
END_REGION

REGION Network 38: Totalizer FT-12.02 HotWater Homomixer
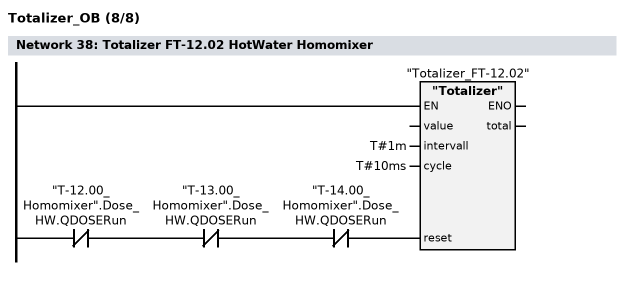
   RUNG wire#powerrail
      "Totalizer_FT-12.02"(reset := wire#w1, value :=, intervall := T#1m, cycle := T#10ms, total =>)
   END_RUNG
   RUNG wire#powerrail
      I_Contact( "T-12.00_Homomixer".Dose_HW.QDOSERun )
      I_Contact( "T-13.00_Homomixer".Dose_HW.QDOSERun )
      I_Contact( "T-14.00_Homomixer".Dose_HW.QDOSERun )
   END_RUNG wire#w1
   // the same network as SCL:
   "Totalizer_FT-12.02"(intervall := T#1m,   // "Totalizer"
                        cycle := T#10ms,
                        reset := NOT "T-12.00_Homomixer".Dose_HW.QDOSERun AND NOT "T-13.00_Homomixer".Dose_HW.QDOSERun AND NOT "T-14.00_Homomixer".Dose_HW.QDOSERun);
END_REGION
END_ORGANIZATION_BLOCK
